FUNCTION_BLOCK VerticalAct
VAR_INPUT
END_VAR
VAR_OUTPUT
	Raise	: BOOL;
	Raised	: BOOL;
	Lowered	: BOOL;
	
END_VAR
VAR
END_VAR

METHOD mLowered : BOOL
VAR_INPUT
END_VAR
END_METHOD

METHOD mRaise : BOOL
VAR_INPUT
END_VAR
//IF ActInputs.Lowered AND ActInputs.Closed THEN (Faulty)
//	Raise	:= ActOutputs.Raise := TRUE;
//END_IF

Raise	:= TRUE;
END_METHOD

METHOD mRaised : BOOL
VAR_INPUT
END_VAR
END_METHOD

PROPERTY pLowered : BOOL
GET
pLowered := Lowered;
END_GET
SET
Lowered := pLowered;
END_SET
END_PROPERTY

PROPERTY pRaise : BOOL
GET
pRaise	:= Raise;
END_GET
SET
Raise	:= pRaise;
END_SET
END_PROPERTY

PROPERTY pRaised : BOOL
GET
pRaised := Raised;
END_GET
SET
Raised := pRaised;
END_SET
END_PROPERTY

END_FUNCTION_BLOCK

(* stored: Version 1.1.0.1, ProductVersion 3.1.4024.9
   POU VerticalAct: Id {b1e5f042-2a3c-4ede-b9a2-0c96d2b214e8}, SpecialFunc None
   Method mLowered: Id {61dc1d1c-e0a0-4745-92df-c122aafdab83}
   Method mRaise: Id {6e30b7e4-a35d-4cd6-a4ec-2261cee925a9}
   Method mRaised: Id {8a76852e-2198-4159-868a-8dbba841f2de}
   Property pLowered: Id {26abcb61-6cbb-4cad-a6d3-97ed43afad3d}
   Get Get: Id {2479cd0a-b4fe-4f54-9d08-045dd52bf6bf}
   Set Set: Id {a5af9486-a2c8-4b38-95a6-ac76b8a4ebb5}
   Property pRaise: Id {96a8ba01-74c1-4db6-97cb-f7d5a98067f7}
   Get Get: Id {547bb4a2-d0a8-4664-9fa3-7ed85ca956ab}
   Set Set: Id {62457140-efcb-4254-a8a1-1b7cdef35bf8}
   Property pRaised: Id {fbfbbb30-2010-46d0-85ba-ef2a4de095fa}
   Get Get: Id {4073d389-6dd8-47e8-9b6c-71f6fb08d612}
   Set Set: Id {3cbee1f5-49a9-46ce-bfa9-629f52c94277} *)
